Staubli VAL3: RobotStatusMsg.pjx

Parameters version=s7.7.2 stackSize=5000 millimeterUnit=true
Program file=start.pgx
Program file=stop.pgx
Data file=RobotStatusMsg.dtx
Type name=RobotStatus path=../RobotStatus/RobotStatus.pjx
Type name=Prefix path=../Prefix/Prefix.pjx
Type name=Header path=../Header/Header.pjx
Type name=Body path=../Body/Body.pjx
